// TIA Portal V18 export
FUNCTION_BLOCK "Xray_related_FB"   // FB56, FBD
{ S7_Optimized_Access := 'TRUE' }
VERSION : 0.1
// stored: AutoNumber true, IsIECCheckEnabled false, IsRetainMemResEnabled false, MemoryReserve 100, SetENOAutomatically false, UDAEnableTagReadback false
   VAR_OUTPUT
      fpd_power : Bool;
   END_VAR
BEGIN

REGION Network 1
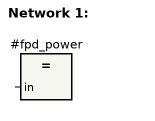
   #fpd_power := TRUE;
END_REGION
END_FUNCTION_BLOCK
